{attribute 'GeneratedUsingTerminal: EL3423-0000-0020'}
{attribute addProperty BoxType "EL3423-0000-0020"}
{attribute addProperty Id "Apparent_EnergyAT %I*LINT8"}
{attribute addProperty CRC "1266626580"}
{attribute addProperty Size "8"}
TYPE Total_Apparent_Reduced_4B7F3014 EXTENDS InputBase_8311D824 :
STRUCT
	{attribute addProperty Name "Apparent_Energy"}
	Apparent_Energy AT %I* : LINT;
END_STRUCT
END_TYPE

(* stored: Version 1.2.0.0, ProductVersion 3.1.4024.9
   DUT Total_Apparent_Reduced_4B7F3014: Id {136ea620-5afa-4ba7-a50c-fbb9f756f6f2} *)
